% RSLogix 500 project multipositionServoApplication.RSS, saved by version 8.30.00.16 %
PROJECT "UNTITLED"    % processor: Bul.1763 MicroLogix 1100 Series B %

PROGRAM FILES
  LAD 2   4 rungs
  LAD 3 "I/O"  7 rungs
  LAD 4 "CTRL LOGIC"  14 rungs
  LAD 5 "STAGES"  6 rungs

DATA FILES
  O0 OUTPUT  4 elements
  I1 INPUT  6 elements
  S2 STATUS  66 elements
  B3 BINARY  11 elements
  T4 TIMER  3 elements
  C5 COUNTER  1 elements
  R6 CONTROL  1 elements
  N7 INTEGER  4 elements
  F8 FLOAT  1 elements

LADDER 2
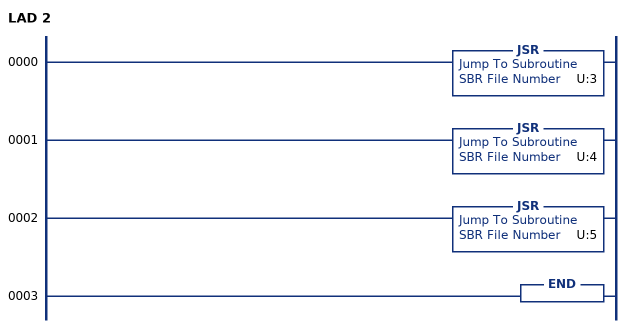
% Rung: 0 %
SOR JSR U:3 EOR
% Rung: 1 %
SOR JSR U:4 EOR
% Rung: 2 %
SOR JSR U:5 EOR
% Rung: 3 %
SOR END EOR

LADDER 3 "I/O"
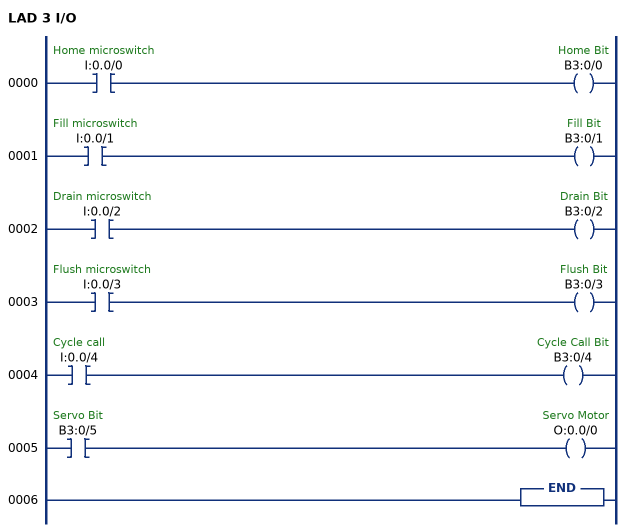
% Rung: 0 %
SOR XIC I:0.0/0 OTE B3:0/0 EOR
%   I:0.0/0  "Home microswitch" %
%   B3:0/0  "Home Bit" %
% Rung: 1 %
SOR XIC I:0.0/1 OTE B3:0/1 EOR
%   I:0.0/1  "Fill microswitch" %
%   B3:0/1  "Fill Bit" %
% Rung: 2 %
SOR XIC I:0.0/2 OTE B3:0/2 EOR
%   I:0.0/2  "Drain microswitch" %
%   B3:0/2  "Drain Bit" %
% Rung: 3 %
SOR XIC I:0.0/3 OTE B3:0/3 EOR
%   I:0.0/3  "Flush microswitch" %
%   B3:0/3  "Flush Bit" %
% Rung: 4 %
SOR XIC I:0.0/4 OTE B3:0/4 EOR
%   I:0.0/4  "Cycle call" %
%   B3:0/4  "Cycle Call Bit" %
% Rung: 5 %
SOR XIC B3:0/5 OTE O:0.0/0 EOR
%   B3:0/5  "Servo Bit" %
%   O:0.0/0  "Servo Motor" %
% Rung: 6 %
SOR END EOR

LADDER 4 "CTRL LOGIC"
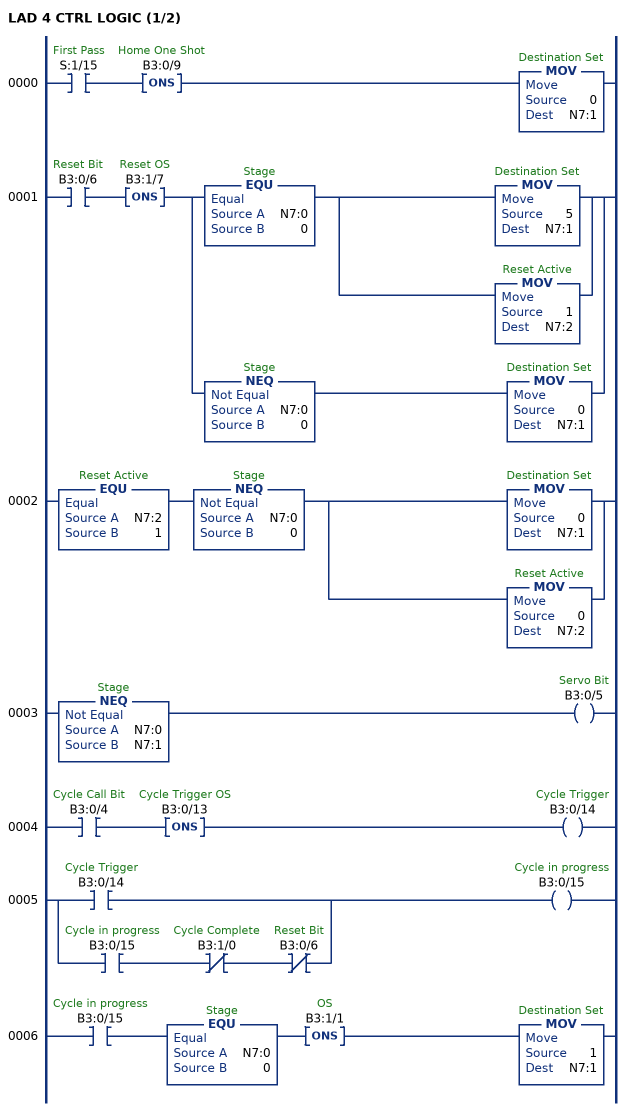
% Rung: 0 %
SOR XIC S:1/15 ONS B3:0/9 MOV 0 N7:1 EOR
%   S:1/15  "First Pass" %
%   B3:0/9  "Home One Shot" %
%   N7:1  "Destination Set" %
% Rung: 1 %
SOR XIC B3:0/6 ONS B3:1/7 BST EQU N7:0 0 BST MOV 5 N7:1 NXB MOV 1 N7:2 BND NXB NEQ N7:0 0 MOV 0 N7:1 BND EOR
%   B3:0/6  "Reset Bit" %
%   B3:1/7  "Reset OS" %
%   N7:0  "Stage" %
%   N7:1  "Destination Set" %
%   N7:2  "Reset Active" %
% Rung: 2 %
SOR EQU N7:2 1 NEQ N7:0 0 BST MOV 0 N7:1 NXB MOV 0 N7:2 BND EOR
%   N7:2  "Reset Active" %
%   N7:0  "Stage" %
%   N7:1  "Destination Set" %
% Rung: 3 %
SOR NEQ N7:0 N7:1 OTE B3:0/5 EOR
%   N7:0  "Stage" %
%   N7:1  "Destination Set" %
%   B3:0/5  "Servo Bit" %
% Rung: 4 %
SOR XIC B3:0/4 ONS B3:0/13 OTE B3:0/14 EOR
%   B3:0/4  "Cycle Call Bit" %
%   B3:0/13  "Cycle Trigger OS" %
%   B3:0/14  "Cycle Trigger" %
% Rung: 5 %
SOR BST XIC B3:0/14 NXB XIC B3:0/15 XIO B3:1/0 XIO B3:0/6 BND OTE B3:0/15 EOR
%   B3:0/14  "Cycle Trigger" %
%   B3:0/15  "Cycle in progress" %
%   B3:1/0  "Cycle Complete" %
%   B3:0/6  "Reset Bit" %
% Rung: 6 %
SOR XIC B3:0/15 EQU N7:0 0 ONS B3:1/1 MOV 1 N7:1 EOR
%   B3:0/15  "Cycle in progress" %
%   N7:0  "Stage" %
%   B3:1/1  "OS" %
%   N7:1  "Destination Set" %

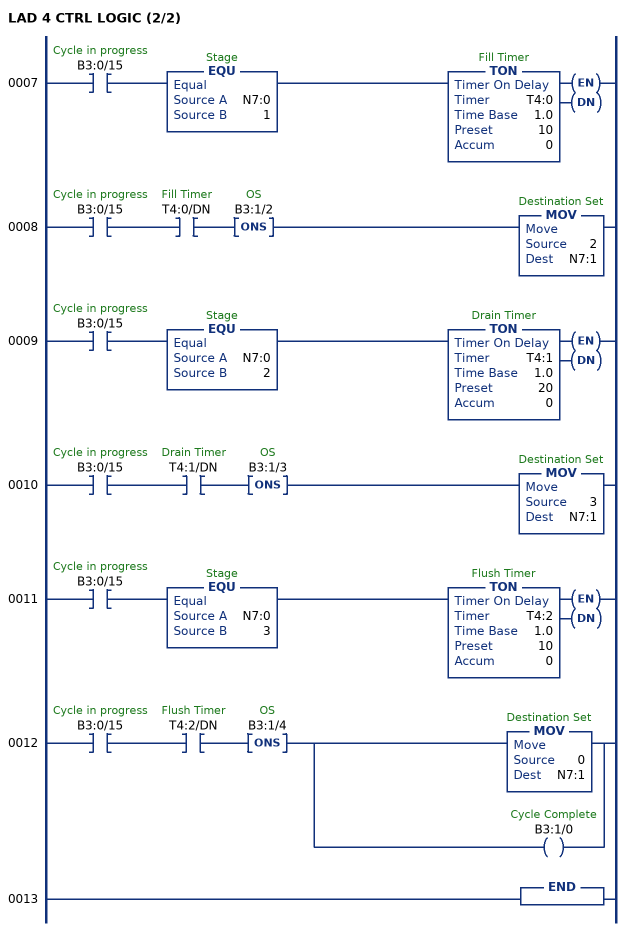
% Rung: 7 %
SOR XIC B3:0/15 EQU N7:0 1 TON T4:0 1.0 10 0 EOR
%   B3:0/15  "Cycle in progress" %
%   N7:0  "Stage" %
%   T4:0  "Fill Timer" %
% Rung: 8 %
SOR XIC B3:0/15 XIC T4:0/DN ONS B3:1/2 MOV 2 N7:1 EOR
%   B3:0/15  "Cycle in progress" %
%   T4:0  "Fill Timer" %
%   B3:1/2  "OS" %
%   N7:1  "Destination Set" %
% Rung: 9 %
SOR XIC B3:0/15 EQU N7:0 2 TON T4:1 1.0 20 0 EOR
%   B3:0/15  "Cycle in progress" %
%   N7:0  "Stage" %
%   T4:1  "Drain Timer" %
% Rung: 10 %
SOR XIC B3:0/15 XIC T4:1/DN ONS B3:1/3 MOV 3 N7:1 EOR
%   B3:0/15  "Cycle in progress" %
%   T4:1/DN  "Drain Timer" %
%   B3:1/3  "OS" %
%   N7:1  "Destination Set" %
% Rung: 11 %
SOR XIC B3:0/15 EQU N7:0 3 TON T4:2 1.0 10 0 EOR
%   B3:0/15  "Cycle in progress" %
%   N7:0  "Stage" %
%   T4:2  "Flush Timer" %
% Rung: 12 %
SOR XIC B3:0/15 XIC T4:2/DN ONS B3:1/4 BST MOV 0 N7:1 NXB OTE B3:1/0 BND EOR
%   B3:0/15  "Cycle in progress" %
%   T4:2/DN  "Flush Timer" %
%   B3:1/4  "OS" %
%   N7:1  "Destination Set" %
%   B3:1/0  "Cycle Complete" %
% Rung: 13 %
SOR END EOR

LADDER 5 "STAGES"
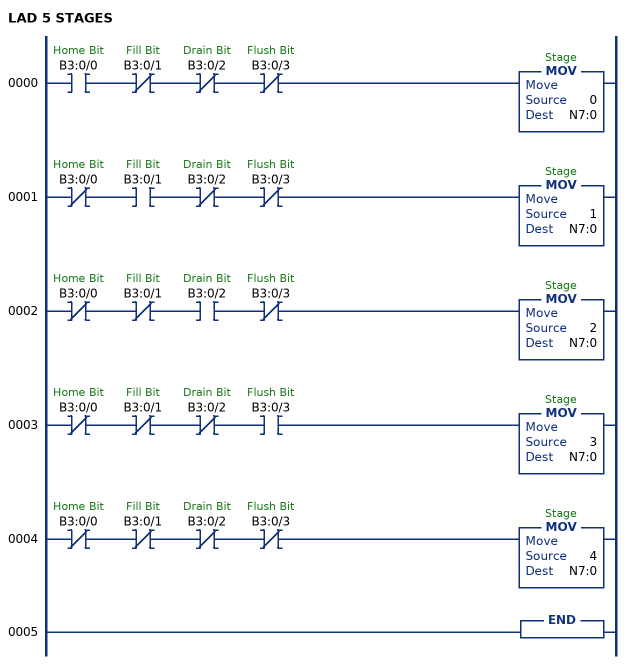
% Rung: 0 %
SOR XIC B3:0/0 XIO B3:0/1 XIO B3:0/2 XIO B3:0/3 MOV 0 N7:0 EOR
%   B3:0/0  "Home Bit" %
%   B3:0/1  "Fill Bit" %
%   B3:0/2  "Drain Bit" %
%   B3:0/3  "Flush Bit" %
%   N7:0  "Stage" %
% Rung: 1 %
SOR XIO B3:0/0 XIC B3:0/1 XIO B3:0/2 XIO B3:0/3 MOV 1 N7:0 EOR
%   B3:0/0  "Home Bit" %
%   B3:0/1  "Fill Bit" %
%   B3:0/2  "Drain Bit" %
%   B3:0/3  "Flush Bit" %
%   N7:0  "Stage" %
% Rung: 2 %
SOR XIO B3:0/0 XIO B3:0/1 XIC B3:0/2 XIO B3:0/3 MOV 2 N7:0 EOR
%   B3:0/0  "Home Bit" %
%   B3:0/1  "Fill Bit" %
%   B3:0/2  "Drain Bit" %
%   B3:0/3  "Flush Bit" %
%   N7:0  "Stage" %
% Rung: 3 %
SOR XIO B3:0/0 XIO B3:0/1 XIO B3:0/2 XIC B3:0/3 MOV 3 N7:0 EOR
%   B3:0/0  "Home Bit" %
%   B3:0/1  "Fill Bit" %
%   B3:0/2  "Drain Bit" %
%   B3:0/3  "Flush Bit" %
%   N7:0  "Stage" %
% Rung: 4 %
SOR XIO B3:0/0 XIO B3:0/1 XIO B3:0/2 XIO B3:0/3 MOV 4 N7:0 EOR
%   B3:0/0  "Home Bit" %
%   B3:0/1  "Fill Bit" %
%   B3:0/2  "Drain Bit" %
%   B3:0/3  "Flush Bit" %
%   N7:0  "Stage" %
% Rung: 5 %
SOR END EOR

OTHER DOCUMENTED ADDRESSES
  B3:0/7  "Initialize command"
  B3:0/8  "Home Trigger"
  B3:0/10  "Fill Trigger"
  B3:0/11  "Drain Trigger"
  B3:0/12  "Flush Trigger"
  B3:1/5  "Startup"
  B3:1/6  "Reset active"
  O:0  "Servo Motor"

DATA TABLE (non-zero values as saved)
DATA T4
% .PRE .ACC %
% T4:0 % 10 0
% T4:1 % 20 0
% T4:2 % 10 0
